TYPE "DecoilersHRot_Status"
VERSION : 0.1
// Block: DecoilersHRot_Status
   STRUCT
      Rotation : ValveMachine_COut;
      Pivot : ValveMachine_COut;
      Traslation : Positioning_DOL_Machine_COut;
      DecoilerX_InLine_CheckNext : Bool;
      Decoiler1_InLine : Bool;
      Decoiler2_InLine : Bool;
      Translation_InPosition : Bool;
   END_STRUCT;

END_TYPE
